(* PLC project Unnamed, Unknown Unnamed 1 *)
(* stored: creationDateTime 2022-08-23T17:04:06, modificationDateTime 2022-08-24T12:04:19 *)

(* Hello World with Ladder Logic Diagram *)
PROGRAM Hello_World
  VAR
    Start_PB AT %I0.0 : BOOL := FALSE;  (* Start Push Button *)
    Stop_PB AT %I0.1 : BOOL := FALSE;  (* Stop Push Button *)
    Motor_Starter AT %Q0.0 : BOOL := FALSE;  (* Soft Motor Starter *)
  END_VAR

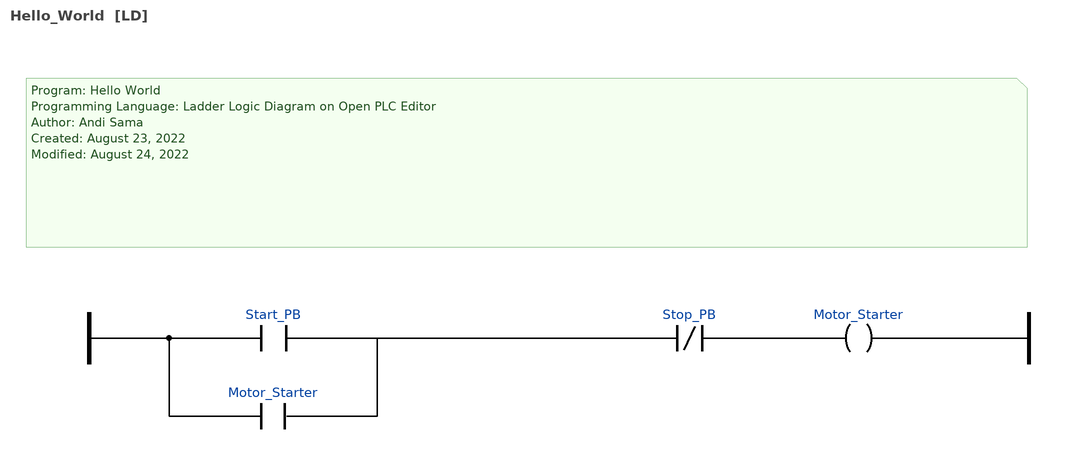
(* LD diagram, written out as Structured Text *)
(* Program: Hello World
Programming Language: Ladder Logic Diagram on Open PLC Editor
Author: Andi Sama
Created: August 23, 2022
Modified: August 24, 2022 *)
Motor_Starter := (Start_PB OR Motor_Starter) AND NOT Stop_PB;
END_PROGRAM

CONFIGURATION Config0
  RESOURCE Res0 ON PLC
    TASK task0(INTERVAL := T#20ms, PRIORITY := 0);
    PROGRAM instance0 WITH task0 : Hello_World;
  END_RESOURCE
END_CONFIGURATION
